// Brief: Slave Arm Joint1-3 decelerate to stop
FUNCTION_BLOCK PUBLIC FB_SlaveCtrlStop EXTENDS FB_SlaveArmCtrlBase
VAR
	// stop motion is terminated after set time period
	m_maxStopPeriod :LREAL := 0.12;
	
	// deceleration period 
	m_decPeriod :LREAL := 0.1;
END_VAR

// override this function in each exact controller
METHOD PROTECTED calcCmdJntPos : BOOL
VAR_IN_OUT CONSTANT
	i_endoscopePose : ST_Frame;
	i_masterStatus :ST_MasterStatus;
	i_setupStatus: ST_SetupStatus;
	i_slaveArm :FB_SlaveArm;
END_VAR

VAR 
	i :INT;
	nextCmdVel :LREAL;
END_VAR
IF m_isFinished THEN
	m_cmdJntVel := g_zeroVec8d;
	m_cmdJntPos := i_slaveArm.curJntPos;
	m_FFJntTrq := g_zeroVec8d;
	RETURN;
END_IF

IF m_timePeriod > m_maxStopPeriod  THEN
	m_isFinished := TRUE;
	RETURN;
END_IF

FOR i := 1 TO 3 DO
	IF m_timePeriod > m_decPeriod THEN
		m_cmdJntVel[i] := 0;
		m_FFJntTrq[i]:=0;
	ELSE
		nextCmdVel := m_cmdJntVel[i] + m_cmdJntAcc[i]*g_slaveArmCtrlCycleTime;
		m_cmdJntPos[i] := m_cmdJntPos[i] + (nextCmdVel + m_cmdJntVel[i])*g_slaveArmCtrlCycleTime/2.0;
		m_cmdJntVel[i] := nextCmdVel;
		m_FFJntTrq[i] :=  i_slaveArm.massMat[i,i] * m_cmdJntAcc[i] ;
	END_IF
END_FOR
END_METHOD

METHOD PUBLIC init : BOOL
VAR_IN_OUT CONSTANT
	i_slaveArm	:FB_SlaveArm;
END_VAR
VAR_IN_OUT 
	r_slaveArmCtrlCmd :ST_SlaveArmCtrlCmds;
END_VAR
VAR
	i:INT;
	maxJntTrq:LREAL;
END_VAR
// check if to hold the command joint position unchanged
m_holdLastCmds := checkToHoldLastCmds(i_slaveArm);
SUPER^.Init(i_slaveArm,r_slaveArmCtrlCmd);

// determine joint deceleration
FOR i:=1 TO 3 DO 
	m_jntOPMode[i] := DriverOPMode_PosTrq;
	m_cmdJntVel[i] := i_slaveArm.curJntVel[i];
	i_slaveArm.m_jntPIDCtrl[i].reset();
	m_cmdJntAcc[i] := -i_slaveArm.curJntVel[i]/m_decPeriod;
END_FOR

// update commands to arm
copyCmds(r_slaveArmCtrlCmd);
END_METHOD

END_FUNCTION_BLOCK

(* stored: Version 1.1.0.1, ProductVersion 3.1.4024.11
   POU FB_SlaveCtrlStop: Id {03e7bf18-07e1-493d-b46e-00a7fc843560}, SpecialFunc None
   Method calcCmdJntPos: Id {5c8aebac-4b88-468e-9571-6f8136c358fb}
   Method init: Id {bd69b8cd-377c-4832-b8a1-80eb64850a03} *)
